TYPE STATE:
    STRUCT
        curTime: REAL;
        dvar_M_Barrier_HW_Barrier_BVH_East_Q_Open: BOOL;
        dvar_M_Barrier_HW_Barrier_BVH_East_Q_Close: BOOL;
        dvar_M_Barrier_HW_TL_BNH_East_Q_Red: BOOL;
        dvar_M_Barrier_HW_TL_BNH_East_Q_Green: BOOL;
        dvar_M_Barrier_HW_TL_BNH_West_Q_Red: BOOL;
        dvar_M_Barrier_HW_TL_BNH_West_Q_Green: BOOL;
        dvar_M_Barrier_HW_TL_BVH_East_Q_Red: BOOL;
        dvar_M_Barrier_HW_TL_BVH_East_Q_Green: BOOL;
        dvar_M_Barrier_HW_TL_BVH_West_Q_Red: BOOL;
        dvar_M_Barrier_HW_TL_BVH_West_Q_Green: BOOL;
        dvar_M_Barrier_SCADA_BarrierOpen: BOOL;
        dvar_M_Barrier_SCADA_BarrierClose: BOOL;
        dvar_M_Barrier_SCADA_BarrierStop: BOOL;
        dvar_M_Barrier_SCADA_DownstreamTLRed: BOOL;
        dvar_M_Barrier_SCADA_DownstreamTLGreen: BOOL;
        dvar_M_Barrier_SCADA_UpstreamTLRed: BOOL;
        dvar_M_Barrier_SCADA_UpstreamTLGreen: BOOL;
        dvar_M_Barrier_SCADA: INT;
        dvar_M_North_HW_EnteringTL_BNH_East_Q_Red: BOOL;
        dvar_M_North_HW_EnteringTL_BNH_East_Q_Green: BOOL;
        dvar_M_North_HW_EnteringTL_BNH_East_Q_RedRed: BOOL;
        dvar_M_North_HW_EnteringTL_BNH_West_Q_Red: BOOL;
        dvar_M_North_HW_EnteringTL_BNH_West_Q_Green: BOOL;
        dvar_M_North_HW_EnteringTL_BNH_West_Q_RedRed: BOOL;
        dvar_M_North_HW_EnteringTL_BVH_East_Q_Red: BOOL;
        dvar_M_North_HW_EnteringTL_BVH_East_Q_Green: BOOL;
        dvar_M_North_HW_EnteringTL_BVH_East_Q_RedRed: BOOL;
        dvar_M_North_HW_EnteringTL_BVH_West_Q_Red: BOOL;
        dvar_M_North_HW_EnteringTL_BVH_West_Q_Green: BOOL;
        dvar_M_North_HW_EnteringTL_BVH_West_Q_RedRed: BOOL;
        dvar_M_North_HW_Gate_BNH_East_Q_Open: BOOL;
        dvar_M_North_HW_Gate_BNH_East_Q_Close: BOOL;
        dvar_M_North_HW_Gate_BNH_West_Q_Open: BOOL;
        dvar_M_North_HW_Gate_BNH_West_Q_Close: BOOL;
        dvar_M_North_HW_Gate_BVH_East_Q_Open: BOOL;
        dvar_M_North_HW_Gate_BVH_East_Q_Close: BOOL;
        dvar_M_North_HW_Gate_BVH_West_Q_Open: BOOL;
        dvar_M_North_HW_Gate_BVH_West_Q_Close: BOOL;
        dvar_M_North_HW_LeavingTL_BNH_East_Q_Red: BOOL;
        dvar_M_North_HW_LeavingTL_BNH_East_Q_Green: BOOL;
        dvar_M_North_HW_LeavingTL_BNH_West_Q_Red: BOOL;
        dvar_M_North_HW_LeavingTL_BNH_West_Q_Green: BOOL;
        dvar_M_North_HW_LeavingTL_BVH_East_Q_Red: BOOL;
        dvar_M_North_HW_LeavingTL_BVH_East_Q_Green: BOOL;
        dvar_M_North_HW_LeavingTL_BVH_West_Q_Red: BOOL;
        dvar_M_North_HW_LeavingTL_BVH_West_Q_Green: BOOL;
        dvar_M_North_HW_Paddle_BNH_East_Q_Open: BOOL;
        dvar_M_North_HW_Paddle_BNH_East_Q_Close: BOOL;
        dvar_M_North_HW_Paddle_BNH_West_Q_Open: BOOL;
        dvar_M_North_HW_Paddle_BNH_West_Q_Close: BOOL;
        dvar_M_North_HW_Paddle_BVH_East_Q_Open: BOOL;
        dvar_M_North_HW_Paddle_BVH_East_Q_Close: BOOL;
        dvar_M_North_HW_Paddle_BVH_West_Q_Open: BOOL;
        dvar_M_North_HW_Paddle_BVH_West_Q_Close: BOOL;
        dvar_M_North_SCADA_DownstreamGateOpen: BOOL;
        dvar_M_North_SCADA_DownstreamGateClose: BOOL;
        dvar_M_North_SCADA_DownstreamGateStop: BOOL;
        dvar_M_North_SCADA_DownstreamPaddleOpen: BOOL;
        dvar_M_North_SCADA_DownstreamPaddleClose: BOOL;
        dvar_M_North_SCADA_DownstreamPaddleStop: BOOL;
        dvar_M_North_SCADA_DownstreamEnteringTLRedRed: BOOL;
        dvar_M_North_SCADA_DownstreamEnteringTLRed: BOOL;
        dvar_M_North_SCADA_DownstreamEnteringTLRedGreen: BOOL;
        dvar_M_North_SCADA_DownstreamEnteringTLGreen: BOOL;
        dvar_M_North_SCADA_DownstreamLeavingTLRed: BOOL;
        dvar_M_North_SCADA_DownstreamLeavingTLGreen: BOOL;
        dvar_M_North_SCADA_UpstreamGateOpen: BOOL;
        dvar_M_North_SCADA_UpstreamGateClose: BOOL;
        dvar_M_North_SCADA_UpstreamGateStop: BOOL;
        dvar_M_North_SCADA_UpstreamPaddleOpen: BOOL;
        dvar_M_North_SCADA_UpstreamPaddleClose: BOOL;
        dvar_M_North_SCADA_UpstreamPaddleStop: BOOL;
        dvar_M_North_SCADA_UpstreamEnteringTLRedRed: BOOL;
        dvar_M_North_SCADA_UpstreamEnteringTLRed: BOOL;
        dvar_M_North_SCADA_UpstreamEnteringTLRedGreen: BOOL;
        dvar_M_North_SCADA_UpstreamEnteringTLGreen: BOOL;
        dvar_M_North_SCADA_UpstreamLeavingTLRed: BOOL;
        dvar_M_North_SCADA_UpstreamLeavingTLGreen: BOOL;
        dvar_M_North_SCADA: INT;
        dvar_M_South_HW_EnteringTL_BNH_East_Q_Red: BOOL;
        dvar_M_South_HW_EnteringTL_BNH_East_Q_Green: BOOL;
        dvar_M_South_HW_EnteringTL_BNH_East_Q_RedRed: BOOL;
        dvar_M_South_HW_EnteringTL_BNH_West_Q_Red: BOOL;
        dvar_M_South_HW_EnteringTL_BNH_West_Q_Green: BOOL;
        dvar_M_South_HW_EnteringTL_BNH_West_Q_RedRed: BOOL;
        dvar_M_South_HW_EnteringTL_BVH_East_Q_Red: BOOL;
        dvar_M_South_HW_EnteringTL_BVH_East_Q_Green: BOOL;
        dvar_M_South_HW_EnteringTL_BVH_East_Q_RedRed: BOOL;
        dvar_M_South_HW_EnteringTL_BVH_West_Q_Red: BOOL;
        dvar_M_South_HW_EnteringTL_BVH_West_Q_Green: BOOL;
        dvar_M_South_HW_EnteringTL_BVH_West_Q_RedRed: BOOL;
        dvar_M_South_HW_Gate_BNH_East_Q_Open: BOOL;
        dvar_M_South_HW_Gate_BNH_East_Q_Close: BOOL;
        dvar_M_South_HW_Gate_BNH_West_Q_Open: BOOL;
        dvar_M_South_HW_Gate_BNH_West_Q_Close: BOOL;
        dvar_M_South_HW_Gate_BVH_East_Q_Open: BOOL;
        dvar_M_South_HW_Gate_BVH_East_Q_Close: BOOL;
        dvar_M_South_HW_Gate_BVH_West_Q_Open: BOOL;
        dvar_M_South_HW_Gate_BVH_West_Q_Close: BOOL;
        dvar_M_South_HW_LeavingTL_BNH_East_Q_Red: BOOL;
        dvar_M_South_HW_LeavingTL_BNH_East_Q_Green: BOOL;
        dvar_M_South_HW_LeavingTL_BNH_West_Q_Red: BOOL;
        dvar_M_South_HW_LeavingTL_BNH_West_Q_Green: BOOL;
        dvar_M_South_HW_LeavingTL_BVH_East_Q_Red: BOOL;
        dvar_M_South_HW_LeavingTL_BVH_East_Q_Green: BOOL;
        dvar_M_South_HW_LeavingTL_BVH_West_Q_Red: BOOL;
        dvar_M_South_HW_LeavingTL_BVH_West_Q_Green: BOOL;
        dvar_M_South_HW_Paddle_BNH_East_Q_Open: BOOL;
        dvar_M_South_HW_Paddle_BNH_East_Q_Close: BOOL;
        dvar_M_South_HW_Paddle_BNH_West_Q_Open: BOOL;
        dvar_M_South_HW_Paddle_BNH_West_Q_Close: BOOL;
        dvar_M_South_HW_Paddle_BVH_East_Q_Open: BOOL;
        dvar_M_South_HW_Paddle_BVH_East_Q_Close: BOOL;
        dvar_M_South_HW_Paddle_BVH_West_Q_Open: BOOL;
        dvar_M_South_HW_Paddle_BVH_West_Q_Close: BOOL;
        dvar_M_South_SCADA_DownstreamGateOpen: BOOL;
        dvar_M_South_SCADA_DownstreamGateClose: BOOL;
        dvar_M_South_SCADA_DownstreamGateStop: BOOL;
        dvar_M_South_SCADA_DownstreamPaddleOpen: BOOL;
        dvar_M_South_SCADA_DownstreamPaddleClose: BOOL;
        dvar_M_South_SCADA_DownstreamPaddleStop: BOOL;
        dvar_M_South_SCADA_DownstreamEnteringTLRedRed: BOOL;
        dvar_M_South_SCADA_DownstreamEnteringTLRed: BOOL;
        dvar_M_South_SCADA_DownstreamEnteringTLRedGreen: BOOL;
        dvar_M_South_SCADA_DownstreamEnteringTLGreen: BOOL;
        dvar_M_South_SCADA_DownstreamLeavingTLRed: BOOL;
        dvar_M_South_SCADA_DownstreamLeavingTLGreen: BOOL;
        dvar_M_South_SCADA_UpstreamGateOpen: BOOL;
        dvar_M_South_SCADA_UpstreamGateClose: BOOL;
        dvar_M_South_SCADA_UpstreamGateStop: BOOL;
        dvar_M_South_SCADA_UpstreamPaddleOpen: BOOL;
        dvar_M_South_SCADA_UpstreamPaddleClose: BOOL;
        dvar_M_South_SCADA_UpstreamPaddleStop: BOOL;
        dvar_M_South_SCADA_UpstreamEnteringTLRedRed: BOOL;
        dvar_M_South_SCADA_UpstreamEnteringTLRed: BOOL;
        dvar_M_South_SCADA_UpstreamEnteringTLRedGreen: BOOL;
        dvar_M_South_SCADA_UpstreamEnteringTLGreen: BOOL;
        dvar_M_South_SCADA_UpstreamLeavingTLRed: BOOL;
        dvar_M_South_SCADA_UpstreamLeavingTLGreen: BOOL;
        dvar_M_South_SCADA: INT;
        dvar_M_sup_Barrier_Barrier_Actuator: INT;
        dvar_M_sup_Barrier_Barrier_Sensor: INT;
        dvar_M_sup_Barrier_Commands: INT;
        dvar_M_sup_Barrier_Downstream_TLs_East_Actuator: INT;
        dvar_M_sup_Barrier_Downstream_TLs_East_SensorG: INT;
        dvar_M_sup_Barrier_Downstream_TLs_East_SensorR: INT;
        dvar_M_sup_Barrier_Downstream_TLs_West_Actuator: INT;
        dvar_M_sup_Barrier_Downstream_TLs_West_SensorG: INT;
        dvar_M_sup_Barrier_Downstream_TLs_West_SensorR: INT;
        dvar_M_sup_Barrier_EmergencyStop: INT;
        dvar_M_sup_Barrier_Upstream_TLs_East_Actuator: INT;
        dvar_M_sup_Barrier_Upstream_TLs_East_SensorG: INT;
        dvar_M_sup_Barrier_Upstream_TLs_East_SensorR: INT;
        dvar_M_sup_Barrier_Upstream_TLs_West_Actuator: INT;
        dvar_M_sup_Barrier_Upstream_TLs_West_SensorG: INT;
        dvar_M_sup_Barrier_Upstream_TLs_West_SensorR: INT;
        dvar_M_sup_North_Commands: INT;
        dvar_M_sup_North_Downstream_EnteringTLs_East_Actuator: INT;
        dvar_M_sup_North_Downstream_EnteringTLs_East_SensorG: INT;
        dvar_M_sup_North_Downstream_EnteringTLs_East_SensorR1: INT;
        dvar_M_sup_North_Downstream_EnteringTLs_East_SensorR2: INT;
        dvar_M_sup_North_Downstream_EnteringTLs_West_Actuator: INT;
        dvar_M_sup_North_Downstream_EnteringTLs_West_SensorG: INT;
        dvar_M_sup_North_Downstream_EnteringTLs_West_SensorR1: INT;
        dvar_M_sup_North_Downstream_EnteringTLs_West_SensorR2: INT;
        dvar_M_sup_North_Downstream_EqualWaterSensor: INT;
        dvar_M_sup_North_Downstream_Gates_East_Actuator: INT;
        dvar_M_sup_North_Downstream_Gates_East_Sensor: INT;
        dvar_M_sup_North_Downstream_Gates_West_Actuator: INT;
        dvar_M_sup_North_Downstream_Gates_West_Sensor: INT;
        dvar_M_sup_North_Downstream_LeavingTLs_East_Actuator: INT;
        dvar_M_sup_North_Downstream_LeavingTLs_East_SensorG: INT;
        dvar_M_sup_North_Downstream_LeavingTLs_East_SensorR: INT;
        dvar_M_sup_North_Downstream_LeavingTLs_West_Actuator: INT;
        dvar_M_sup_North_Downstream_LeavingTLs_West_SensorG: INT;
        dvar_M_sup_North_Downstream_LeavingTLs_West_SensorR: INT;
        dvar_M_sup_North_Downstream_Paddles_East_Actuator: INT;
        dvar_M_sup_North_Downstream_Paddles_East_Sensor: INT;
        dvar_M_sup_North_Downstream_Paddles_West_Actuator: INT;
        dvar_M_sup_North_Downstream_Paddles_West_Sensor: INT;
        dvar_M_sup_North_EmergencyStop: INT;
        dvar_M_sup_North_Upstream_EnteringTLs_East_Actuator: INT;
        dvar_M_sup_North_Upstream_EnteringTLs_East_SensorG: INT;
        dvar_M_sup_North_Upstream_EnteringTLs_East_SensorR1: INT;
        dvar_M_sup_North_Upstream_EnteringTLs_East_SensorR2: INT;
        dvar_M_sup_North_Upstream_EnteringTLs_West_Actuator: INT;
        dvar_M_sup_North_Upstream_EnteringTLs_West_SensorG: INT;
        dvar_M_sup_North_Upstream_EnteringTLs_West_SensorR1: INT;
        dvar_M_sup_North_Upstream_EnteringTLs_West_SensorR2: INT;
        dvar_M_sup_North_Upstream_EqualWaterSensor: INT;
        dvar_M_sup_North_Upstream_Gates_East_Actuator: INT;
        dvar_M_sup_North_Upstream_Gates_East_Sensor: INT;
        dvar_M_sup_North_Upstream_Gates_West_Actuator: INT;
        dvar_M_sup_North_Upstream_Gates_West_Sensor: INT;
        dvar_M_sup_North_Upstream_LeavingTLs_East_Actuator: INT;
        dvar_M_sup_North_Upstream_LeavingTLs_East_SensorG: INT;
        dvar_M_sup_North_Upstream_LeavingTLs_East_SensorR: INT;
        dvar_M_sup_North_Upstream_LeavingTLs_West_Actuator: INT;
        dvar_M_sup_North_Upstream_LeavingTLs_West_SensorG: INT;
        dvar_M_sup_North_Upstream_LeavingTLs_West_SensorR: INT;
        dvar_M_sup_North_Upstream_Paddles_East_Actuator: INT;
        dvar_M_sup_North_Upstream_Paddles_East_Sensor: INT;
        dvar_M_sup_North_Upstream_Paddles_West_Actuator: INT;
        dvar_M_sup_North_Upstream_Paddles_West_Sensor: INT;
        dvar_M_sup_South_Commands: INT;
        dvar_M_sup_South_Downstream_EnteringTLs_East_Actuator: INT;
        dvar_M_sup_South_Downstream_EnteringTLs_East_SensorG: INT;
        dvar_M_sup_South_Downstream_EnteringTLs_East_SensorR1: INT;
        dvar_M_sup_South_Downstream_EnteringTLs_East_SensorR2: INT;
        dvar_M_sup_South_Downstream_EnteringTLs_West_Actuator: INT;
        dvar_M_sup_South_Downstream_EnteringTLs_West_SensorG: INT;
        dvar_M_sup_South_Downstream_EnteringTLs_West_SensorR1: INT;
        dvar_M_sup_South_Downstream_EnteringTLs_West_SensorR2: INT;
        dvar_M_sup_South_Downstream_EqualWaterSensor: INT;
        dvar_M_sup_South_Downstream_Gates_East_Actuator: INT;
        dvar_M_sup_South_Downstream_Gates_East_Sensor: INT;
        dvar_M_sup_South_Downstream_Gates_West_Actuator: INT;
        dvar_M_sup_South_Downstream_Gates_West_Sensor: INT;
        dvar_M_sup_South_Downstream_LeavingTLs_East_Actuator: INT;
        dvar_M_sup_South_Downstream_LeavingTLs_East_SensorG: INT;
        dvar_M_sup_South_Downstream_LeavingTLs_East_SensorR: INT;
        dvar_M_sup_South_Downstream_LeavingTLs_West_Actuator: INT;
        dvar_M_sup_South_Downstream_LeavingTLs_West_SensorG: INT;
        dvar_M_sup_South_Downstream_LeavingTLs_West_SensorR: INT;
        dvar_M_sup_South_Downstream_Paddles_East_Actuator: INT;
        dvar_M_sup_South_Downstream_Paddles_East_Sensor: INT;
        dvar_M_sup_South_Downstream_Paddles_West_Actuator: INT;
        dvar_M_sup_South_Downstream_Paddles_West_Sensor: INT;
        dvar_M_sup_South_EmergencyStop: INT;
        dvar_M_sup_South_Upstream_EnteringTLs_East_Actuator: INT;
        dvar_M_sup_South_Upstream_EnteringTLs_East_SensorG: INT;
        dvar_M_sup_South_Upstream_EnteringTLs_East_SensorR1: INT;
        dvar_M_sup_South_Upstream_EnteringTLs_East_SensorR2: INT;
        dvar_M_sup_South_Upstream_EnteringTLs_West_Actuator: INT;
        dvar_M_sup_South_Upstream_EnteringTLs_West_SensorG: INT;
        dvar_M_sup_South_Upstream_EnteringTLs_West_SensorR1: INT;
        dvar_M_sup_South_Upstream_EnteringTLs_West_SensorR2: INT;
        dvar_M_sup_South_Upstream_EqualWaterSensor: INT;
        dvar_M_sup_South_Upstream_Gates_East_Actuator: INT;
        dvar_M_sup_South_Upstream_Gates_East_Sensor: INT;
        dvar_M_sup_South_Upstream_Gates_West_Actuator: INT;
        dvar_M_sup_South_Upstream_Gates_West_Sensor: INT;
        dvar_M_sup_South_Upstream_LeavingTLs_East_Actuator: INT;
        dvar_M_sup_South_Upstream_LeavingTLs_East_SensorG: INT;
        dvar_M_sup_South_Upstream_LeavingTLs_East_SensorR: INT;
        dvar_M_sup_South_Upstream_LeavingTLs_West_Actuator: INT;
        dvar_M_sup_South_Upstream_LeavingTLs_West_SensorG: INT;
        dvar_M_sup_South_Upstream_LeavingTLs_West_SensorR: INT;
        dvar_M_sup_South_Upstream_Paddles_East_Actuator: INT;
        dvar_M_sup_South_Upstream_Paddles_East_Sensor: INT;
        dvar_M_sup_South_Upstream_Paddles_West_Actuator: INT;
        dvar_M_sup_South_Upstream_Paddles_West_Sensor: INT;
    END_STRUCT;
END_TYPE
